{attribute 'qualified_only'}
{attribute 'strict'}
TYPE E_WarehouseState :
(
    IDLE    := 0,
    RUNNING := 1,
    PAUSED  := 2,
    FAULT   := 99
);
END_TYPE

(* stored: Version 1.1.0.1, ProductVersion 3.1.4024.16
   DUT E_WarehouseState: Id {f6a7b8c9-d0e1-2345-f012-678901234567} *)
